FUNCTION "_checkVelocity" : LReal
TITLE = Function:Check velocity
{ S7_Optimized_Access := 'TRUE' }
AUTHOR : cyanezf
FAMILY : Controller/Util
NAME : _checkVelocity
VERSION : 1.0

   VAR_INPUT
      MIN_VELOCITY : LReal;   // Min velocity
      MAX_VELOCITY : LReal;   // Max velocity
      inVelocity : LReal;   // Cururent velocity
   END_VAR

BEGIN
(*--

# Log
| version | date | author | description |
|:-------:|:----:|:------:|:------------|
| v1.0 | 2023-12-12 | cyanezf | First version |

# Dependencies
| Dependency |
|:-----------|

# Description
This function checks `inVelocity` variable is between `MIN_VELOCITY` and `MAX_VELOCITY` and returns
the velocity in range if overflow is detected.

#
_Use [Markdown Live Preview](https://markdownlivepreview.com/) to watch this doc._
--*)

	IF #inVelocity > 0.0 THEN

	  IF #inVelocity > #MAX_VELOCITY THEN
	    #_checkVelocity := #MAX_VELOCITY;
	  ELSIF #inVelocity < #MIN_VELOCITY THEN
	    #_checkVelocity := #MIN_VELOCITY;
	  ELSE
	    #_checkVelocity:= #inVelocity;
	  END_IF;

	ELSIF #inVelocity < 0.0 THEN

	  IF ABS(#inVelocity) > #MAX_VELOCITY THEN
	    #_checkVelocity := - #MAX_VELOCITY;
	  ELSIF ABS(#inVelocity) < #MIN_VELOCITY THEN
	    #_checkVelocity := - #MIN_VELOCITY;
	  ELSE
	    #_checkVelocity := #inVelocity;
	  END_IF;

	ELSE

	  #_checkVelocity := #inVelocity;

	END_IF;

	// Save RLO
	ENO := true;

END_FUNCTION

